// TIA Portal V21 export
FUNCTION "Main Portate" : Void   // FC19, LAD
{ S7_Optimized_Access := 'TRUE' }
// stored: SetENOAutomatically false
   VAR_TEMP
      AnalogNotUsed : "Std_VarGestAnalog";
      ImpulsoNotUsed : Bool;
      Appo_StructAnalog : "Std_VarGestAnalog";
   END_VAR
BEGIN
END_FUNCTION
